{attribute 'qualified_only'}
{attribute 'strict'}
TYPE E_CRYO_BIN_ACT_FEEDBACK_STATE :
(
	OFF		:= 0,
	ON	 	:= 1,
	ERROR	:= 2
);
END_TYPE

(* stored: Version 1.1.0.1, ProductVersion 3.1.4024.9
   DUT E_CRYO_BIN_ACT_FEEDBACK_STATE: Id {a55c1633-7d71-4e51-afd3-c501c8644ab2} *)
